{attribute 'qualified_only'}
VAR_GLOBAL
    xRunRequest     : BOOL;
    xHomeSensor     : BOOL;
    xProductPresent : BOOL;
    rTargetVolume   : LREAL := 250.0;   // ml
END_VAR

(* stored: Version 1.1.0.1, ProductVersion 3.1.4024.0
   GVL GVL_Machine: Id {6d13f8b2-40ae-4c97-85d1-e2093ba4f7c6} *)
